PROGRAM MAIN
VAR
END_VAR

//PRG_RCC();

END_PROGRAM

(* stored: Version 1.1.0.1, ProductVersion 3.1.4024.12
   POU MAIN: Id {a8605b09-14c1-42af-ad44-9e0837ea999a}, SpecialFunc None *)
